FUNCTION_BLOCK SkillMagazineController (* Basic Function Block Type *)
  (* Standard: 61499-2 *)
  (* Version 0.0, 2/16/2024, midxav, Template *)
  PACKAGE Main;
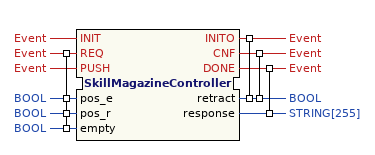
  EVENT_INPUT
    INIT; (* Initialization Request *)
    REQ WITH pos_e, pos_r, empty; (* Normal Execution Request *)
    PUSH;
  END_EVENT
  EVENT_OUTPUT
    INITO WITH retract; (* Initialization Confirm *)
    CNF WITH retract; (* Execution Confirmation *)
    DONE WITH response;
  END_EVENT
  VAR_INPUT
    pos_e : BOOL; (* Input event qualifier *)
    pos_r : BOOL;
    empty : BOOL;
  END_VAR
  VAR_OUTPUT
    retract : BOOL; (* Output event qualifier *)
    response : STRING[255];
  END_VAR
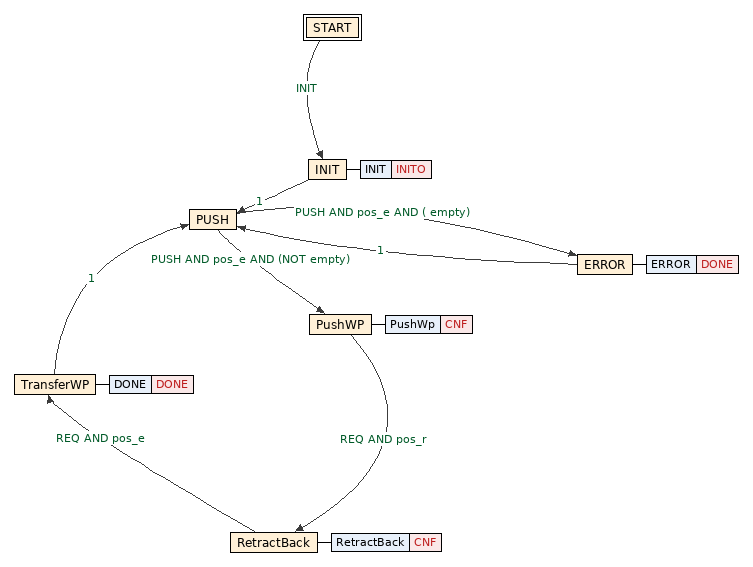
  EC_STATES
    START; (* Initial State *)
    INIT : INIT -> INITO; (* Initialization *)
    PushWP : PushWp -> CNF;
    RetractBack : RetractBack -> CNF;
    TransferWP : DONE -> DONE;
    PUSH;
    ERROR : ERROR -> DONE;
  END_STATES
  EC_TRANSITIONS
    START TO INIT := INIT;
    PUSH TO PushWP := PUSH AND pos_e AND (NOT empty);
    PushWP TO RetractBack := REQ AND pos_r;
    RetractBack TO TransferWP := REQ AND pos_e;
    TransferWP TO PUSH := 1;
    INIT TO PUSH := 1;
    PUSH TO ERROR := PUSH AND pos_e AND ( empty);
    ERROR TO PUSH := 1;
  END_TRANSITIONS
  ALGORITHM INIT IN ST: (* Initialization algorithm *)
retract := FALSE;
  END_ALGORITHM
  ALGORITHM PushWp IN ST:
retract := TRUE;
  END_ALGORITHM
  ALGORITHM RetractBack IN ST:
retract := FALSE;
  END_ALGORITHM
  ALGORITHM DONE IN ST:
response:='WP PUSHED';
  END_ALGORITHM
  ALGORITHM ERROR IN ST:
response:='MAG IS EMPTY';
  END_ALGORITHM
END_FUNCTION_BLOCK
